(* IEC 61131-3 sources: ArfBotOS/Codesys-4/ArfBotOS.fbsdev/Application.iecapp^/FUN/FB_CommandProcessor.fb.st^/protected, 11 files *)

(* ---- M_Aborting.meth.st ---- *)
METHOD PROTECTED M_Aborting : BOOL

CASE _SeqAborting OF
	0:
		_ProcessMoveCommand.M_Abort();
		_ProcessPauseCommand.M_Abort();
		//_ProcessInputCommand.M_Abort();
		_ProcessOutputCommand.M_Abort();
		_ProcessVisionCommand.M_Abort();
		_ProcessVarSetCommand.M_Abort();
		_ProcessCncCommand.M_Abort();
		_ProcessLogicCommand.M_Abort();
		_SeqAborting := _SeqAborting + 1;
	1:
		IF _ProcessMoveCommand.PropCurrentState = PACK_ML.State.Aborted
			AND _ProcessPauseCommand.PropCurrentState = PACK_ML.State.Aborted
			//AND _ProcessInputCommand.PropCurrentState = PACK_ML.State.Aborted
			AND _ProcessOutputCommand.PropCurrentState = PACK_ML.State.Aborted
			AND _ProcessVisionCommand.PropCurrentState = PACK_ML.State.Aborted
			AND _ProcessVarSetCommand.PropCurrentState = PACK_ML.State.Aborted
			AND _ProcessCncCommand.PropCurrentState = PACK_ML.State.Aborted
			AND _ProcessLogicCommand.PropCurrentState = PACK_ML.State.Aborted THEN
				_SeqAborting := 0;
				SUPER^.M_StateComplete();
		END_IF

END_CASE

(*IF ItfActiveModule <> 0 THEN
	ItfActiveModule.M_Abort();
	IF ItfActiveModule.PropCurrentState = PACK_ML.State.Aborted THEN
		SUPER^.M_StateComplete();
	END_IF
ELSE
	SUPER^.M_StateComplete();
END_IF*)
END_METHOD

(* ---- M_Execute.meth.st ---- *)
METHOD PROTECTED M_Execute : BOOL
VAR
    _ErrorDescription: STRING;
END_VAR

// here we want to execute our commands/jobs/etc and set completed when done.
//
CASE _SeqMain OF
  	_STEP_DONE:
		_SeqMain := _STEP_IDLE;

	_STEP_IDLE:
		// hang out here until called to run
		_CurrentCmdIdx := 0;
		SUPER^.M_StateComplete();

	_STEP_CMD: //
		IF NOT Enable THEN
			_SeqMain := _STEP_DONE;
            _ErrorDescription := '';
            IF NOT GVL_App.Enable THEN
                _ErrorDescription := 'Robot not enabled';
            END_IF
            IF NOT PersistentVars.Flags[GVL_App.HOME_COMPLETE].Value THEN
                _ErrorDescription := CONCAT(_ErrorDescription, ' | Robot not homed');
            END_IF
            IF GVL_App.xActiveAlarm THEN
                _ErrorDescription := CONCAT(_ErrorDescription, ' | Active alarms exist');
            END_IF
            IF _ErrorDescription = '' THEN
                _ErrorDescription := 'Not enabled';
            END_IF
            _M_Error(Description := _ErrorDescription);

		ELSIF _CurrentCmdIdx <= GVL_App.PROG_CMDS_ARR_END AND _CurrentCmdIdx >= GVL_App.PROG_CMDS_ARR_BEG THEN
			//
			IF _Commands[_CurrentCmdIdx].CommandType = DUT_CommandType.Disabled THEN
				// want to increment here so that we can disable some commands
				// in the program and it continue to execute
				_CurrentCmdIdx := _CurrentCmdIdx + 1;
				_SeqMain := _STEP_CMD;

			ELSE
				CASE _Commands[_CurrentCmdIdx].CommandType OF
					DUT_CommandType.MoveCommand: //
						StatusText := 'Move Command in Progress';
						ItfActiveProcessorUnitMode := _ProcessMoveCommand.ItfUnitMode;
						ItfActiveModule := _ProcessMoveCommand;
						_ProcessMoveCommand.Command := _Commands[_CurrentCmdIdx].CommandString;
						ItfActiveModule.M_Start();

					DUT_CommandType.PauseCommand: //
						StatusText := 'Pause Command in Progress';
						ItfActiveProcessorUnitMode := _ProcessPauseCommand.ItfUnitMode;
						ItfActiveModule := _ProcessPauseCommand;
						_ProcessPauseCommand.Command := _Commands[_CurrentCmdIdx].CommandString;
						ItfActiveModule.M_Start();

					DUT_CommandType.InputCommand: //
						StatusText := 'Input Command in Progress';
						//ActiveUnitMode := _ProcessInputCommand.ItfUnitMode;
						//ItfActiveModule := _ProcessInputCommand;
						//_ProcessInputCommand.Command := _Commands[_CurrentCmdIdx].CommandString;
						//ItfActiveModule.M_Start();

					DUT_CommandType.OutputCommand: //
						StatusText := 'Output Command in Progress';
						ItfActiveProcessorUnitMode := _ProcessOutputCommand.ItfUnitMode;
						ItfActiveModule := _ProcessOutputCommand;
						_ProcessOutputCommand.Command := _Commands[_CurrentCmdIdx].CommandString;
						ItfActiveModule.M_Start();

					DUT_CommandType.VisionCommand: //
						StatusText := 'Vision Command in Progress';
						ItfActiveProcessorUnitMode := _ProcessVisionCommand.ItfUnitMode;
						ItfActiveModule := _ProcessVisionCommand;
						_ProcessVisionCommand.Command := _Commands[_CurrentCmdIdx].CommandString;
						ItfActiveModule.M_Start();

					DUT_CommandType.VarSetCommand: //
						StatusText := 'VarSet Command in Progress';
						ItfActiveProcessorUnitMode := _ProcessVarsetCommand.ItfUnitMode;
						ItfActiveModule := _ProcessVarsetCommand;
						_ProcessVarsetCommand.Command := _Commands[_CurrentCmdIdx].CommandString;
						ItfActiveModule.M_Start();

					DUT_CommandType.CncCommand: //
						StatusText := 'CNC Command in Progress';
						ItfActiveProcessorUnitMode := _ProcessCncCommand.ItfUnitMode;
						ItfActiveModule := _ProcessCncCommand;
						_ProcessCncCommand.Command := _Commands[_CurrentCmdIdx].CommandString;
						ItfActiveModule.M_Start();

					DUT_CommandType.LogicCommand: //
						StatusText := 'Logic Command in Progress';
						ItfActiveProcessorUnitMode := _ProcessLogicCommand.ItfUnitMode;
						ItfActiveModule := _ProcessLogicCommand;
						_ProcessLogicCommand.Command := _Commands[_CurrentCmdIdx].CommandString;
						ItfActiveModule.M_Start();

				ELSE
					_SeqMain := _STEP_CMD;

				END_CASE

				// wait for executing
				IF ItfActiveModule.PropCurrentState = PACK_ML.State.Execute THEN
					_ActiveCommand := _Commands[_CurrentCmdIdx];
					_CurrentCmdIdx := _CurrentCmdIdx + 1;
					_SeqMain := _STEP_WAIT;
				END_IF
			END_IF

		ELSE
			_SeqMain := _STEP_DONE;
		END_IF

	_STEP_WAIT: // wait for command to finish
		//
		IF _ProcessorDoneRtrig.Q THEN
			_SeqMain := _STEP_CMD;
		END_IF
		//
		IF ItfActiveModule.PropError THEN
			SUPER^._UnitMode.Suspend();
			_SeqMain := _STEP_ERR;
		END_IF

	_STEP_ERR: //

END_CASE

// watch for rising edge of idle state. this was done for all processors since
// the vision processor runs in a separate task and isnt guaranteed to start in the same
// PLC scan.
_ProcessorDoneRtrig(clk:=ItfActiveProcessorUnitMode.CurrentState = PACK_ML.State.Idle);
END_METHOD

(* ---- M_Holding.meth.st ---- *)
METHOD PROTECTED M_Holding : BOOL

IF ItfActiveModule <> 0 THEN
	ItfActiveModule.M_Hold();
	IF ItfActiveModule.PropCurrentState = PACK_ML.State.Held THEN
		SUPER^.M_StateComplete();
	END_IF
ELSE
	SUPER^.M_StateComplete();
END_IF
END_METHOD

(* ---- M_Idle.meth.st ---- *)
METHOD PROTECTED M_Idle : BOOL

// in this state, we want to reset all the function blocks and hang out
_SeqMain := _STEP_IDLE;
_SeqAborting := 0;
_SeqClearing := 0;
_SeqResetting := 0;
END_METHOD

(* ---- M_Resetting.meth.st ---- *)
METHOD PROTECTED M_Resetting : BOOL

CASE _SeqResetting OF
	0:
		_ProcessMoveCommand.M_Home();
		_ProcessPauseCommand.M_Home();
		//_ProcessInputCommand.M_Home();
		_ProcessOutputCommand.M_Home();
		_ProcessVisionCommand.M_Home();
		_ProcessVarSetCommand.M_Home();
		_ProcessCncCommand.M_Home();
		_ProcessLogicCommand.M_Home();
        StatusText := 'Resetting';
		_SeqResetting := _SeqResetting + 1;
	1:
		IF _ProcessMoveCommand.PropCurrentState = PACK_ML.State.Idle
			AND _ProcessPauseCommand.PropCurrentState = PACK_ML.State.Idle
			//AND _ProcessInputCommand.PropCurrentState = PACK_ML.State.Idle
			AND _ProcessOutputCommand.PropCurrentState = PACK_ML.State.Idle
			AND _ProcessVisionCommand.PropCurrentState = PACK_ML.State.Idle
			AND _ProcessVarSetCommand.PropCurrentState = PACK_ML.State.Idle
			AND _ProcessCncCommand.PropCurrentState = PACK_ML.State.Idle
			AND _ProcessLogicCommand.PropCurrentState = PACK_ML.State.Idle THEN
				_SeqResetting := 0;
                StatusText := 'Idle';
				SUPER^.M_StateComplete();
		END_IF

END_CASE

SUPER^.M_Reset();

(*IF ItfActiveModule <> 0 THEN
	CASE _Seq OF
		0:
			IF NOT ItfActiveModule.PropCurrentState = PACK_ML.State.Idle THEN
				ItfActiveModule.M_Home();
				_Seq := 1;
			ELSE
				SUPER^.M_StateComplete();
			END_IF
		1:
			IF ItfActiveModule.PropCurrentState = PACK_ML.State.Idle THEN
				_Seq := 0;
			END_IF

	END_CASE

ELSE
	SUPER^.M_StateComplete();
	_Seq := 0;

END_IF*)
END_METHOD

(* ---- M_SetPackML.meth.st ---- *)
METHOD PROTECTED M_SetPackML : BOOL

// SUPER already does this but the default is eInitialState:=PACK_ML.State.Idle
// and we want PACK_ML.State.Aborted for the Orchestrator
SUPER^._UnitMode(sName := 'Command Processor',
				eInitialState := PACK_ML.State.Aborted,
				xActive := TRUE);
END_METHOD

(* ---- M_Starting.meth.st ---- *)
METHOD PROTECTED M_Starting : BOOL

// here we want to clear things and get ready for the execute state
// we can consider this the "INIT" state
_SeqMain := _STEP_CMD;
SUPER^._TimeoutTimer.PT := T#0MS; // timeout is ignored if set to 0
SUPER^.M_StateComplete();
END_METHOD

(* ---- M_Stopping.meth.st ---- *)
METHOD PROTECTED M_Stopping : BOOL

IF ItfActiveModule <> 0 THEN
	ItfActiveModule.M_Stop();
	IF ItfActiveModule.PropCurrentState = PACK_ML.State.Idle
		OR ItfActiveModule.PropCurrentState = PACK_ML.State.Stopped
		OR ItfActiveModule.PropCurrentState = PACK_ML.State.Aborted
		OR ItfActiveModule.PropCurrentState = PACK_ML.State.Complete THEN
			SUPER^.M_StateComplete();
	END_IF

ELSE
	SUPER^.M_StateComplete();

END_IF
END_METHOD

(* ---- M_Suspending.meth.st ---- *)
METHOD PROTECTED M_Suspending : BOOL

IF ItfActiveModule <> 0 THEN
	IF ItfActiveModule.PropCurrentState = PACK_ML.State.Execute THEN
		ItfActiveModule.M_Hold();
		IF ItfActiveModule.PropCurrentState = PACK_ML.State.Held THEN
			SUPER^.M_StateComplete();
		END_IF
	ELSE
		SUPER^.M_StateComplete();
	END_IF

ELSE
	SUPER^.M_StateComplete();

END_IF
END_METHOD

(* ---- M_UnHolding.meth.st ---- *)
METHOD PROTECTED M_Unholding : BOOL

//
IF ItfActiveModule <> 0 THEN
	ItfActiveModule.M_Start();
	IF ItfActiveModule.PropCurrentState = PACK_ML.State.Execute THEN
		SUPER^.M_StateComplete();
	END_IF

ELSE
	SUPER^.M_StateComplete();

END_IF

//
_SeqMain := _STEP_WAIT;
END_METHOD

(* ---- M_UnSuspending.meth.st ---- *)
METHOD PROTECTED M_UnSuspending : BOOL

//
IF ItfActiveModule <> 0 THEN
	ItfActiveModule.M_Start();
	IF ItfActiveModule.PropCurrentState = PACK_ML.State.Execute THEN
		SUPER^.M_StateComplete();
	END_IF

ELSE
	SUPER^.M_StateComplete();

END_IF

//
_SeqMain := _STEP_WAIT;
END_METHOD
